Universal Robots PolyScope program: LocalToMixer.urp

Program LocalToMixer (installation=Youssef directory=/programs/Youssef createdIn=5.9.5.1031259 lastSavedIn=5.9.5.1031259 robotSerialNumber=20215500597)
Calibrated DH parameters: a=[0.000193, -0.066673, -0.391568, -0.000012, 0.00005, 0]; d=[0.162643, -472.05677, 465.132521, 7.058239, 0.099746, 0.099582]; alpha=[1.571116, 0.00089, 0.003862, 1.569269, -1.569248, 0]; deltaTheta=[0, -1.413394, 7.628392, 0.068187, 0, -0.000001]
Robot Program (runOnlyOnce=true)
  MoveJ speed 60 deg/s, acceleration 80 deg/s^2 (useActiveTCP=true) feature=Base
    Waypoint Waypoint_6: TCP in base x=600.329 y=210.742 z=131.498 mm, rx=1.2172 ry=1.1583 rz=1.214 rad; joints [56.082, -110.582, -128.809, -117.898, -32.023, -1.06] deg; TCP offset x=0 y=0 z=191.5 mm, rx=0 ry=0 rz=0 rad
    URCap Gripper (Robotiq_Grippers, Robotiq Inc.) dataModel(position=100.0, force=20.0, speed=5.0, positionInDouble=100.0, forceInDouble=20.0, speedInDouble=5.0, slaveIds=[9], blocking=true)
    Waypoint Waypoint_7: TCP in base x=686.015 y=314.199 z=507.236 mm, rx=1.0724 ry=1.0119 rz=0.973 rad; joints [56.944, -104.036, -80.003, -150.247, -22.204, -33.393] deg
    Waypoint Waypoint_6: TCP in base x=600.329 y=210.742 z=131.498 mm, rx=1.2172 ry=1.1583 rz=1.214 rad; joints [56.082, -110.582, -128.809, -117.898, -32.023, -1.06] deg
    URCap Gripper (Robotiq_Grippers, Robotiq Inc.) dataModel(position=0.0, force=20.0, speed=5.0, positionInDouble=0.0, forceInDouble=20.0, speedInDouble=5.0, slaveIds=[9], blocking=true)
